// TIA Portal V20 export
TYPE "typeSequenceControlNodeJobInterfaceMonitoring"
// stored: Namespace Unit1.Em5
   STRUCT
      busyManPpUnloading { ExternalWritable := 'False'} : Bool;
      doneManPpUnloading { ExternalWritable := 'False'} : Bool;
   END_STRUCT;
END_TYPE
